TYPE ST_MotorCtrl :
STRUCT
	power	: BOOL;
	start	: BOOL;
	stop	: BOOL;
	reset	: BOOL;
	velo 	: INT;
END_STRUCT
END_TYPE

(* stored: Version 1.1.0.1, ProductVersion 3.1.4024.11
   DUT ST_MotorCtrl: Id {ca6227ce-8088-48b3-8958-4e808202a2bb} *)
